Staubli VAL3: home.dtx

public num distance
public num moveType
public num nIndexGun
public num nStop
public num nTcpAction
public num nTime
public string comment
public string instruction
public string sProgram
public bool toStop
public jointRx jJoints
public mdesc nom_speed = {vel=10, tmax=9999, rmax=9999, leave=30, reach=30}
